// Mitsubishi GX Works2 project: C5, T20   PLC: FX1N/FX1NC

PROGRAM MAIN
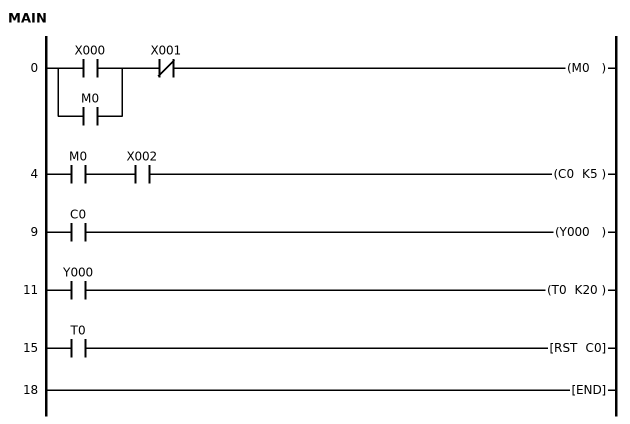
0     LD      X000
      OR      M0
      ANI     X001
      OUT     M0
4     LD      M0
      AND     X002
      OUT     C0 K5
9     LD      C0
      OUT     Y000
11    LD      Y000
      OUT     T0 K20
15    LD      T0
      RST     C0
18    END
END_PROGRAM
